Omron CX-Programmer project 新工程 (CX-Programmer 9.73)

# PLC 新PLC1: CPM2* 

## Global symbols (name address type ; comment)
0.00 BOOL  ; 挡板光电
0.01 BOOL  ; 挡板定位磁开关
0.02 BOOL  ; 一线弹辊光电
0.03 BOOL  ; 一线升降磁开关
0.04 BOOL  ; 二线弹带光电
0.05 BOOL  ; 二线升降磁开关
0.06 BOOL  ; 分砖光电
0.07 BOOL  ; 分砖光电2
10.00 BOOL  ; 接砖辊台
10.01 BOOL  ; 挡板辊台
10.02 BOOL  ; 挡辊高速
10.03 BOOL  ; 一线弹辊
10.04 BOOL  ; 接砖慢速
10.05 BOOL  ; 二线弹辊
10.07 BOOL  ; 一线弹带传动
11.00 BOOL  ; 送砖带
11.01 BOOL  ; 送砖带慢
11.02 BOOL  ; 二线弹带传动
11.03 BOOL  ; 送砖带2
11.04 BOOL  ; 送砖带2慢
11.05 BOOL  ; 转弯带
11.06 BOOL  ; 转弯带2
12.00 BOOL  ; 挡板电机
12.01 BOOL  ; 一线弹带升降
12.02 BOOL  ; 2弹带声升降
12.03 BOOL  ; 连锁输出
1.00 BOOL  ; 总停
1.01 BOOL  ; 总起动
1.02 BOOL  ; 一线开停
1.03 BOOL  ; 关二线
1.04 BOOL  ; 挡板手自
1.06 BOOL  ; 一线联入
1.07 BOOL  ; 二线联入
200.00 BOOL  ; 总起停
201.04 BOOL  ; 下面过砖升分
201.05 BOOL  ; 一线弹辊光电降分
201.06 BOOL  ; 二线弹辊光电降分
201.07 BOOL  ; 挡板升分
20.14 BOOL  ; 一线弹辊光电升分
20.15 BOOL  ; 一线弹辊降分
HR0.00 BOOL  ; 分砖
HR0.01 BOOL  ; 上位锁定
HR0.02 BOOL  ; 分砖2
HR0.03 BOOL  ; 上位锁定2
HR0.04 BOOL  ; 一线弹辊有砖
HR0.05 BOOL  ; 下面过砖
HR0.06 BOOL  ; 一线弹带降
HR0.07 BOOL  ; 二弹辊有砖
HR0.08 BOOL  ; 2弹带降
HR0.09 BOOL  ; 挡板降
HR0.10 BOOL  ; 挡板升
TIM000 BOOL  ; 一线弹带上位
TIM001 BOOL  ; 一线弹带下位
TIM002 BOOL  ; 二线弹带上位
TIM003 BOOL  ; 二线弹带下位
TIM004 BOOL  ; 挡板上位
TIM005 BOOL  ; 挡板下位
TIM016 BOOL  ; 分砖时间
TIM017 BOOL  ; 分砖时间2
TIM018 BOOL  ; 一线弹辊有砖
TIM019 BOOL  ; 挡板延时降
TIM020 BOOL  ; 挡板延时升
TIM021 BOOL  ; 一线弹辊有砖延时
TIM100 BOOL  ; 延时可下降
TIM101 BOOL  ; 延时可下降2
TIM102 BOOL  ; 皮带延时升
TIM103 BOOL  ; 该走一线
TIM104 BOOL  ; 下面过砖时间
TIM105 BOOL  ; 二弹带延时升

## Program 新程序1 (no task)
; 这个PLC程序实现了一个陶瓷厂双釉线干燥窑出窑机系统的控制系统，用于陶瓷生产线的自动化控制。系统通过接砖辊台、挡板辊台、一线弹辊、二线弹辊等设备，将干燥窑内的高温陶瓷坯料接出并分流到两条生产线进行后续加工。 / 系统执行流程： / 1.PLC控制器通过接砖辊台将高温陶瓷坯料从干燥窑内接出。 / 2.挡板辊台启动后进行初步输送。 / 3.工人通过一线开停按钮或二线关闭按钮选择生产线，系统避免转弯带1和转弯带2同时运行以确保分流准确。 / 4.一线运行时，转弯带1和送砖带1启动，分砖光电1信号异常时停止输送以防止坯料堆积。 / 5.二线运行时，转弯带2和送砖带2启动，依赖分砖光电2信号确认坯料状态。 / 6.一线弹带升降运行时需确认一线升降磁开关信号以避免超行程。 / 7.二线弹带升降运行时需确认二线升降磁开关信号。 / 8.挡板电机运行时需确认挡板光电和挡板定位磁开关信号以避免撞击障碍物。 / 9.挡板手自切换启用时，工人可控制挡板上升或下降。 / 10.总停按钮按下时，送砖带1等输出停止以确保安全。 / 11.连锁输出未激活时，送砖带1等输出停止以准备系统。 / 12.一线弹辊和二线弹辊根据一线弹辊光电和二线弹带光电信号调整运行，配合分砖时间定时器1和分砖时间定时器2控制分流。 / 13.挡板电机在手动模式下由挡板上升或下降信号驱动。 / 14.挡板辊台启动时需确认挡板光电信号有效。 / 15.挡板定位磁开关触发后，挡板上位计时开始。 / 16.分砖光电1触发时，分砖动作准备就绪。 / 17.一线弹带升降根据皮带延时升信号启动。 / 18.一线升降磁开关确认后，一线弹带上位计时启动。 / 19.一线开停按钮按下时，转弯带1准备运行。 / 20.总停按钮释放后，总起停信号生效。 / 21.连锁输出激活时，系统进入正常运行状态。

### Section 段1

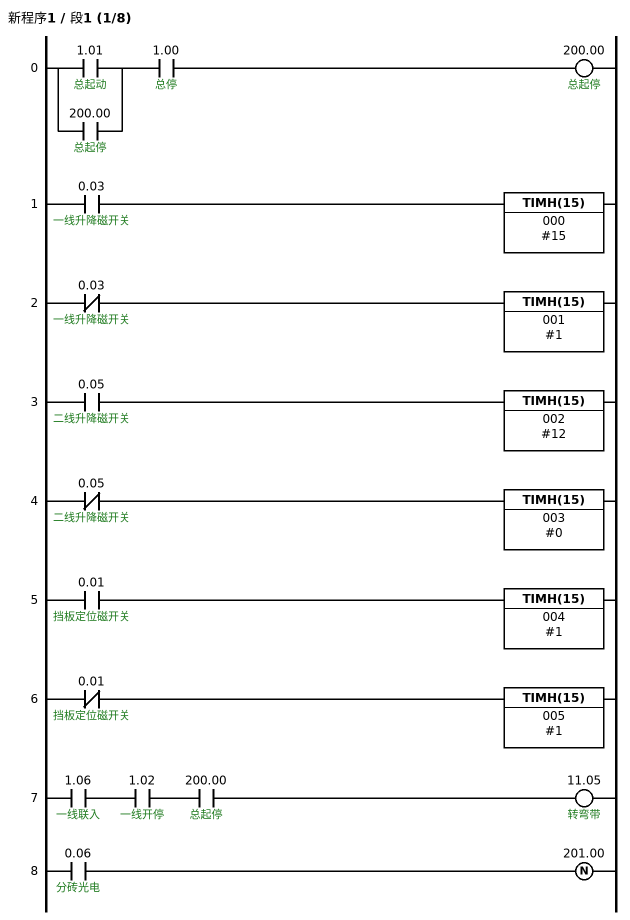
; rung 0
LD 1.01  ; 总起动
OR 200.00  ; 总起停
AND 1.00  ; 总停
OUT 200.00  ; 总起停
; rung 1
LD 0.03  ; 一线升降磁开关
TIMH(15) 000 #15
; rung 2
LDNOT 0.03  ; 一线升降磁开关
TIMH(15) 001 #1
; rung 3
LD 0.05  ; 二线升降磁开关
TIMH(15) 002 #12
; rung 4
LDNOT 0.05  ; 二线升降磁开关
TIMH(15) 003 #0
; rung 5
LD 0.01  ; 挡板定位磁开关
TIMH(15) 004 #1
; rung 6
LDNOT 0.01  ; 挡板定位磁开关
TIMH(15) 005 #1
; rung 7
LD 1.06  ; 一线联入
AND 1.02  ; 一线开停
AND 200.00  ; 总起停
OUT 11.05  ; 转弯带
; rung 8
LD 0.06  ; 分砖光电
DIFD(14) 201.00

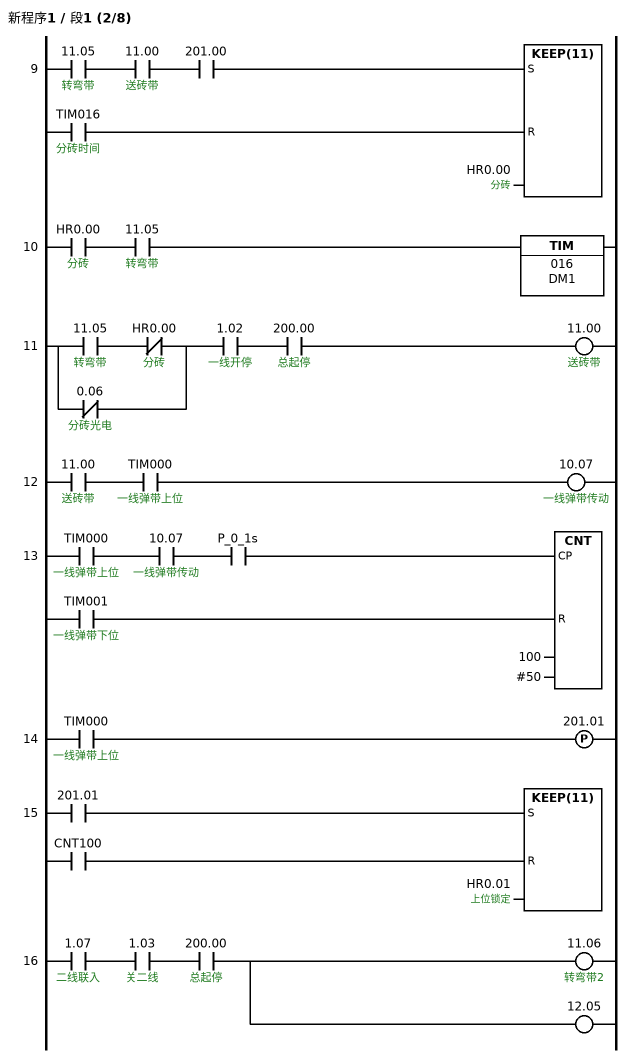
; rung 9
LD 11.05  ; 转弯带
AND 11.00  ; 送砖带
AND 201.00
LD TIM016  ; 分砖时间
KEEP(11) HR0.00  ; 分砖
; rung 10
LD HR0.00  ; 分砖
AND 11.05  ; 转弯带
TIM 016 DM1
; rung 11
LD 11.05  ; 转弯带
ANDNOT HR0.00  ; 分砖
ORNOT 0.06  ; 分砖光电
AND 1.02  ; 一线开停
AND 200.00  ; 总起停
OUT 11.00  ; 送砖带
; rung 12
LD 11.00  ; 送砖带
AND TIM000  ; 一线弹带上位
OUT 10.07  ; 一线弹带传动
; rung 13
LD TIM000  ; 一线弹带上位
AND 10.07  ; 一线弹带传动
AND P_0_1s
LD TIM001  ; 一线弹带下位
CNT 100 #50
; rung 14
LD TIM000  ; 一线弹带上位
DIFU(13) 201.01
; rung 15
LD 201.01
LD CNT100
KEEP(11) HR0.01  ; 上位锁定
; rung 16
LD 1.07  ; 二线联入
AND 1.03  ; 关二线
AND 200.00  ; 总起停
OUT 11.06  ; 转弯带2
OUT 12.05

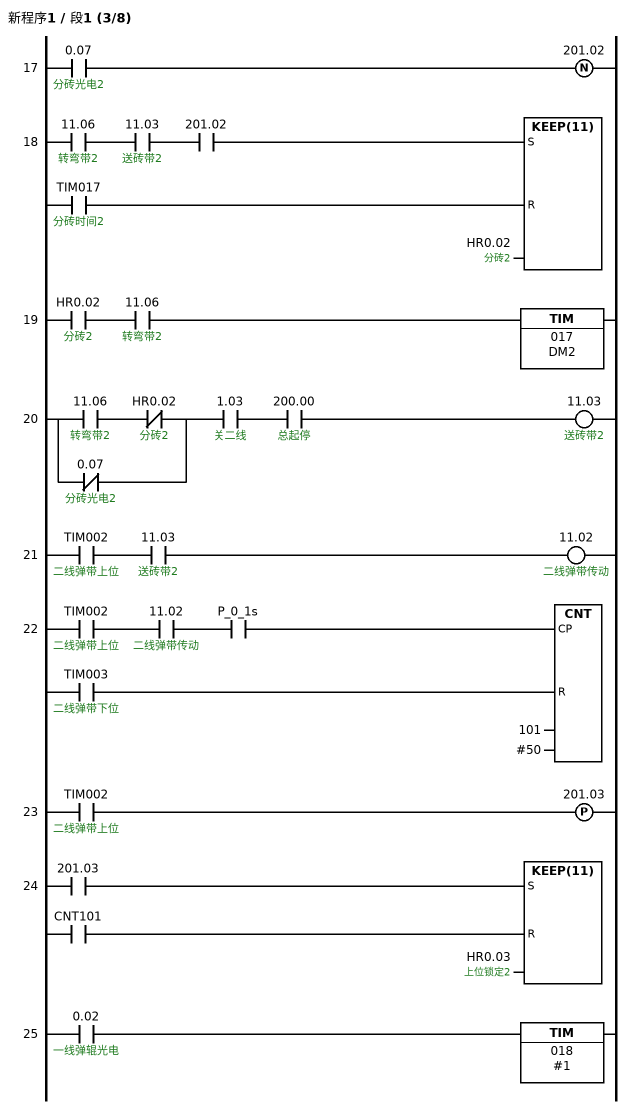
; rung 17
LD 0.07  ; 分砖光电2
DIFD(14) 201.02
; rung 18
LD 11.06  ; 转弯带2
AND 11.03  ; 送砖带2
AND 201.02
LD TIM017  ; 分砖时间2
KEEP(11) HR0.02  ; 分砖2
; rung 19
LD HR0.02  ; 分砖2
AND 11.06  ; 转弯带2
TIM 017 DM2
; rung 20
LD 11.06  ; 转弯带2
ANDNOT HR0.02  ; 分砖2
ORNOT 0.07  ; 分砖光电2
AND 1.03  ; 关二线
AND 200.00  ; 总起停
OUT 11.03  ; 送砖带2
; rung 21
LD TIM002  ; 二线弹带上位
AND 11.03  ; 送砖带2
OUT 11.02  ; 二线弹带传动
; rung 22
LD TIM002  ; 二线弹带上位
AND 11.02  ; 二线弹带传动
AND P_0_1s
LD TIM003  ; 二线弹带下位
CNT 101 #50
; rung 23
LD TIM002  ; 二线弹带上位
DIFU(13) 201.03
; rung 24
LD 201.03
LD CNT101
KEEP(11) HR0.03  ; 上位锁定2
; rung 25
LD 0.02  ; 一线弹辊光电
TIM 018 #1

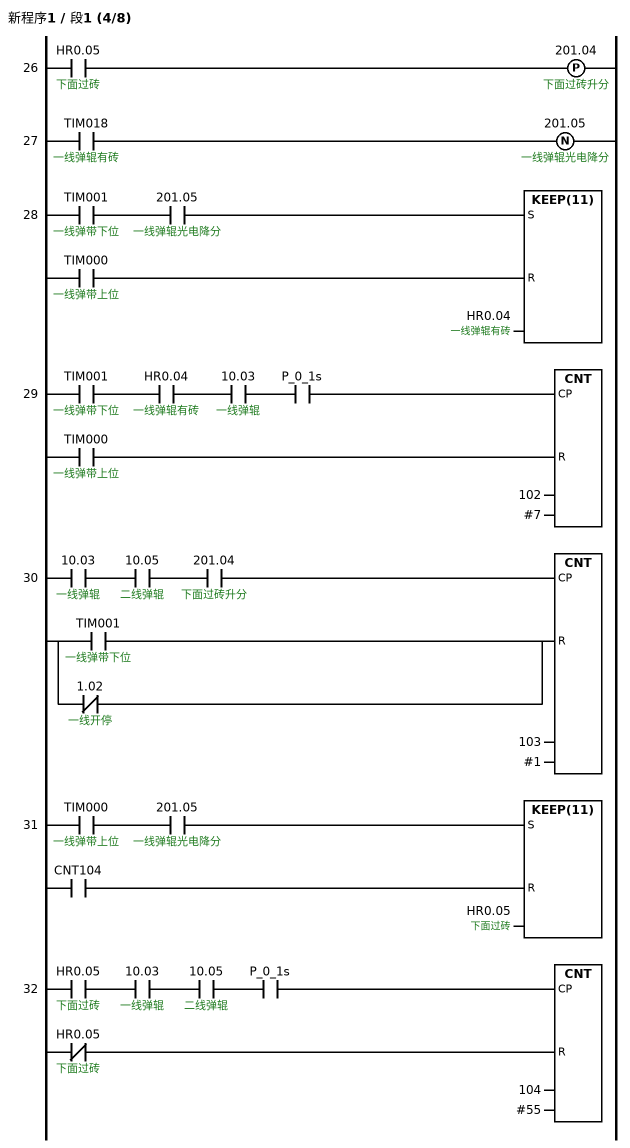
; rung 26
LD HR0.05  ; 下面过砖
DIFU(13) 201.04  ; 下面过砖升分
; rung 27
LD TIM018  ; 一线弹辊有砖
DIFD(14) 201.05  ; 一线弹辊光电降分
; rung 28
LD TIM001  ; 一线弹带下位
AND 201.05  ; 一线弹辊光电降分
LD TIM000  ; 一线弹带上位
KEEP(11) HR0.04  ; 一线弹辊有砖
; rung 29
LD TIM001  ; 一线弹带下位
AND HR0.04  ; 一线弹辊有砖
AND 10.03  ; 一线弹辊
AND P_0_1s
LD TIM000  ; 一线弹带上位
CNT 102 #7
; rung 30
LD 10.03  ; 一线弹辊
AND 10.05  ; 二线弹辊
AND 201.04  ; 下面过砖升分
LD TIM001  ; 一线弹带下位
ORNOT 1.02  ; 一线开停
CNT 103 #1
; rung 31
LD TIM000  ; 一线弹带上位
AND 201.05  ; 一线弹辊光电降分
LD CNT104
KEEP(11) HR0.05  ; 下面过砖
; rung 32
LD HR0.05  ; 下面过砖
AND 10.03  ; 一线弹辊
AND 10.05  ; 二线弹辊
AND P_0_1s
LDNOT HR0.05  ; 下面过砖
CNT 104 #55

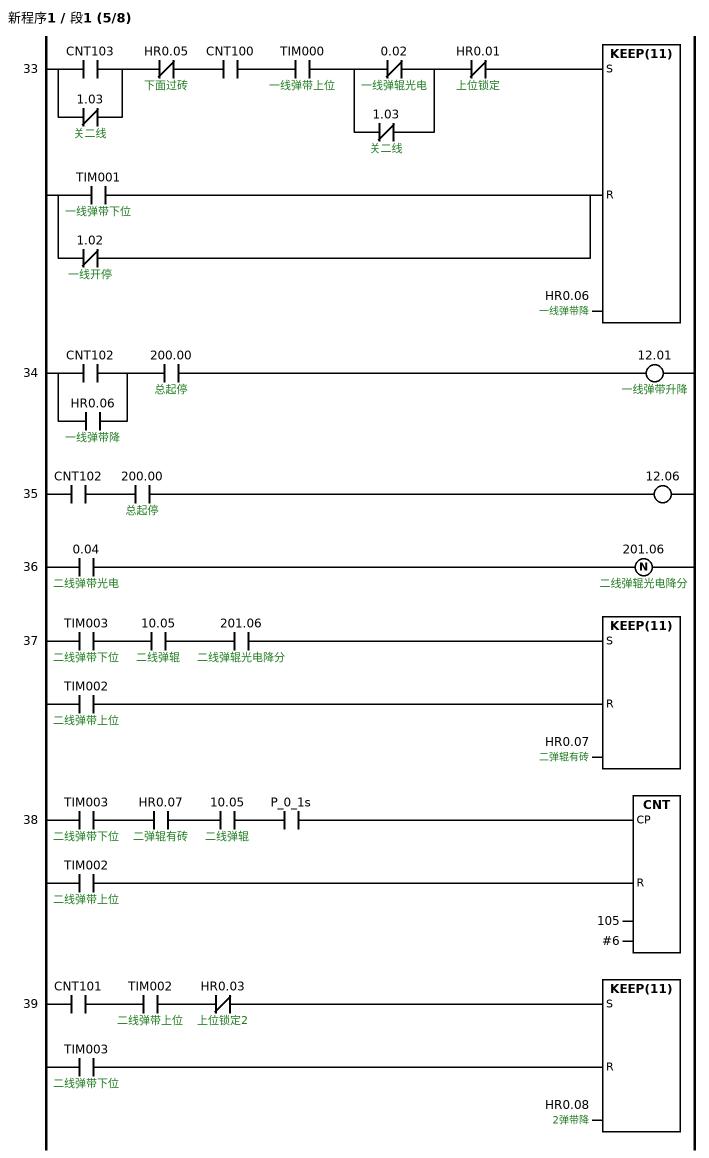
; rung 33
LD CNT103
ORNOT 1.03  ; 关二线
ANDNOT HR0.05  ; 下面过砖
AND CNT100
AND TIM000  ; 一线弹带上位
LDNOT 0.02  ; 一线弹辊光电
ORNOT 1.03  ; 关二线
ANDLD
ANDNOT HR0.01  ; 上位锁定
LD TIM001  ; 一线弹带下位
ORNOT 1.02  ; 一线开停
KEEP(11) HR0.06  ; 一线弹带降
; rung 34
LD CNT102
OR HR0.06  ; 一线弹带降
AND 200.00  ; 总起停
OUT 12.01  ; 一线弹带升降
; rung 35
LD CNT102
AND 200.00  ; 总起停
OUT 12.06
; rung 36
LD 0.04  ; 二线弹带光电
DIFD(14) 201.06  ; 二线弹辊光电降分
; rung 37
LD TIM003  ; 二线弹带下位
AND 10.05  ; 二线弹辊
AND 201.06  ; 二线弹辊光电降分
LD TIM002  ; 二线弹带上位
KEEP(11) HR0.07  ; 二弹辊有砖
; rung 38
LD TIM003  ; 二线弹带下位
AND HR0.07  ; 二弹辊有砖
AND 10.05  ; 二线弹辊
AND P_0_1s
LD TIM002  ; 二线弹带上位
CNT 105 #6
; rung 39
LD CNT101
AND TIM002  ; 二线弹带上位
ANDNOT HR0.03  ; 上位锁定2
LD TIM003  ; 二线弹带下位
KEEP(11) HR0.08  ; 2弹带降

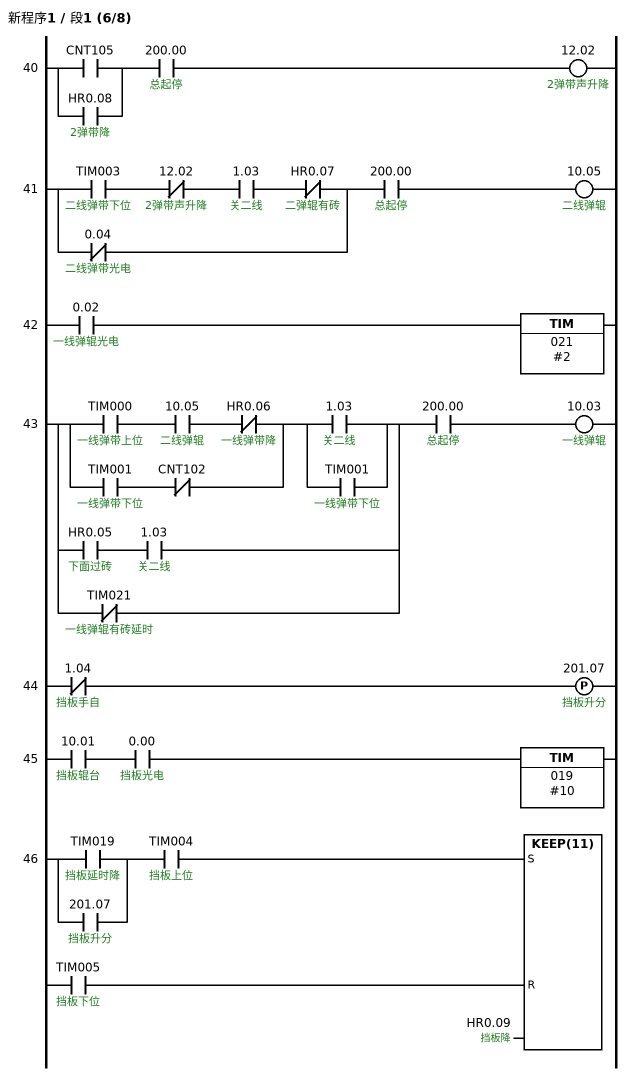
; rung 40
LD CNT105
OR HR0.08  ; 2弹带降
AND 200.00  ; 总起停
OUT 12.02  ; 2弹带声升降
; rung 41
LD TIM003  ; 二线弹带下位
ANDNOT 12.02  ; 2弹带声升降
AND 1.03  ; 关二线
ANDNOT HR0.07  ; 二弹辊有砖
ORNOT 0.04  ; 二线弹带光电
AND 200.00  ; 总起停
OUT 10.05  ; 二线弹辊
; rung 42
LD 0.02  ; 一线弹辊光电
TIM 021 #2
; rung 43
LD TIM000  ; 一线弹带上位
AND 10.05  ; 二线弹辊
ANDNOT HR0.06  ; 一线弹带降
LD TIM001  ; 一线弹带下位
ANDNOT CNT102
ORLD
LD 1.03  ; 关二线
OR TIM001  ; 一线弹带下位
ANDLD
LD HR0.05  ; 下面过砖
AND 1.03  ; 关二线
ORLD
ORNOT TIM021  ; 一线弹辊有砖延时
AND 200.00  ; 总起停
OUT 10.03  ; 一线弹辊
; rung 44
LDNOT 1.04  ; 挡板手自
DIFU(13) 201.07  ; 挡板升分
; rung 45
LD 10.01  ; 挡板辊台
AND 0.00  ; 挡板光电
TIM 019 #10
; rung 46
LD TIM019  ; 挡板延时降
OR 201.07  ; 挡板升分
AND TIM004  ; 挡板上位
LD TIM005  ; 挡板下位
KEEP(11) HR0.09  ; 挡板降

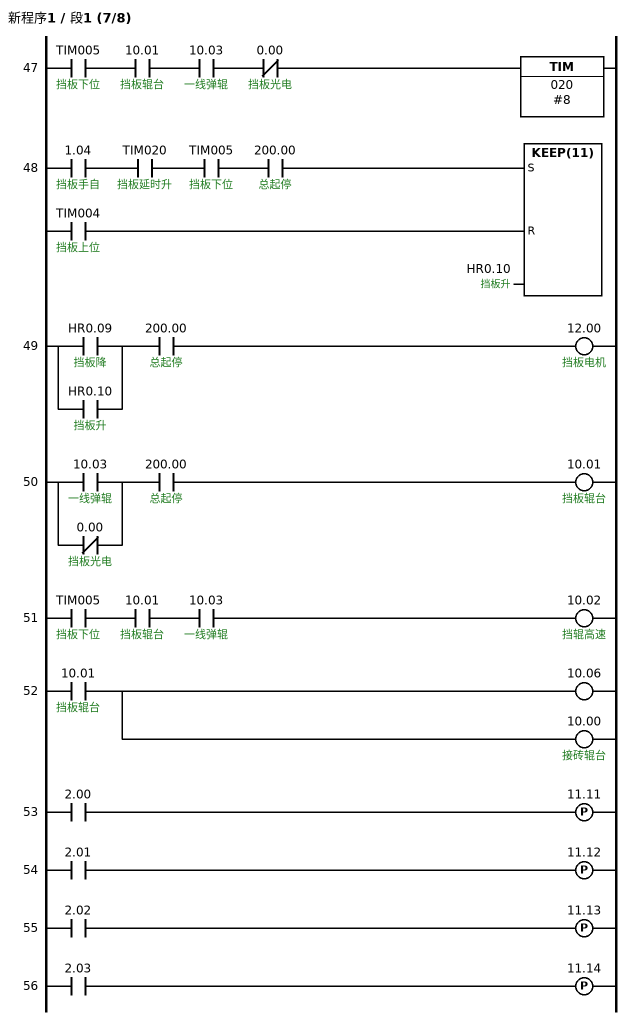
; rung 47
LD TIM005  ; 挡板下位
AND 10.01  ; 挡板辊台
AND 10.03  ; 一线弹辊
ANDNOT 0.00  ; 挡板光电
TIM 020 #8
; rung 48
LD 1.04  ; 挡板手自
AND TIM020  ; 挡板延时升
AND TIM005  ; 挡板下位
AND 200.00  ; 总起停
LD TIM004  ; 挡板上位
KEEP(11) HR0.10  ; 挡板升
; rung 49
LD HR0.09  ; 挡板降
OR HR0.10  ; 挡板升
AND 200.00  ; 总起停
OUT 12.00  ; 挡板电机
; rung 50
LD 10.03  ; 一线弹辊
ORNOT 0.00  ; 挡板光电
AND 200.00  ; 总起停
OUT 10.01  ; 挡板辊台
; rung 51
LD TIM005  ; 挡板下位
AND 10.01  ; 挡板辊台
AND 10.03  ; 一线弹辊
OUT 10.02  ; 挡辊高速
; rung 52
LD 10.01  ; 挡板辊台
OUT 10.06
OUT 10.00  ; 接砖辊台
; rung 53
LD 2.00
DIFU(13) 11.11
; rung 54
LD 2.01
DIFU(13) 11.12
; rung 55
LD 2.02
DIFU(13) 11.13
; rung 56
LD 2.03
DIFU(13) 11.14

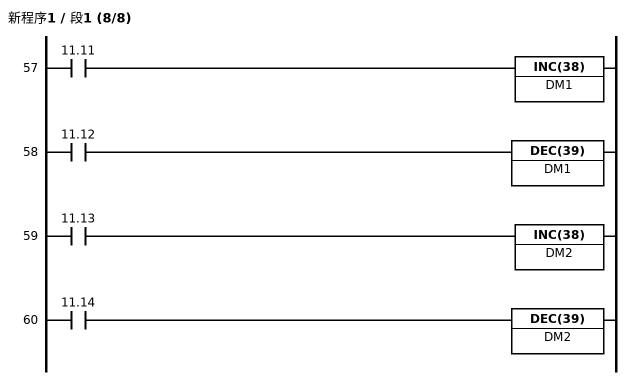
; rung 57
LD 11.11
INC(38) DM1
; rung 58
LD 11.12
DEC(39) DM1
; rung 59
LD 11.13
INC(38) DM2
; rung 60
LD 11.14
DEC(39) DM2
; rung 61
END(01)